// TIA Portal V20 export
TYPE "typeSafetyForcedDoorOpen"
// stored: Access Published, IsFailsafeCompliant true, Namespace Safety
   STRUCT
      Door1OpenMemo : Bool;
      Door2OpenMemo : Bool;
      Door3OpenMemo : Bool;
      Door4OpenMemo : Bool;
      Door5OpenMemo : Bool;
      Door6OpenMemo : Bool;
      Door7OpenMemo : Bool;
      Door8OpenMemo : Bool;
      Door9OpenMemo : Bool;
      Door10OpenMemo : Bool;
      Door1OpenMemoError : Bool;   // Forced Open AUTO SPLICE DOOR
      Door2OpenMemoError : Bool;   // Forced Open UNWIND MAIN DOOR
      Door3OpenMemoError : Bool;   // Forced Open UNWID TOP DOOR
      Door4OpenMemoError : Bool;   // Forced Open UNWIND BOTTOM DOOR
      Door5OpenMemoError : Bool;   // Forced Open STACK TABLE DOOR
      Door6OpenMemoError : Bool;   // Forced Open JR WINDER DOOR
      Door7OpenMemoError : Bool;   // Forced Open ANODE WASTE DOOR
      Door8OpenMemoError : Bool;   // Forced Open STACK TABLE REAR
      Door9OpenMemoError : Bool;   // Forced Open CATHODE WASTE DOOR
      Door10OpenMemoError : Bool;   // Forced Open UNWIND REAR DOOR
      Door1OpenTimeOver : Bool;   // Time Over Open AUTO SPLICE DOOR
      Door2OpenTimeOver : Bool;   // Time Over Open UNWIND MAIN DOOR
      Door3OpenTimeOver : Bool;   // Time Over Open UNWID TOP DOOR
      Door4OpenTimeOver : Bool;   // Time Over Open UNWIND BOTTOM DOOR
      Door5OpenTimeOver : Bool;   // Time Over Open STACK TABLE DOOR
      Door6OpenTimeOver : Bool;   // Time Over Open JR WINDER DOOR
      Door7OpenTimeOver : Bool;   // Time Over Open ANODE WASTE DOOR
      Door8OpenTimeOver : Bool;   // Time Over Open STACK TABLE REAR
      Door9OpenTimeOver : Bool;   // Time Over Open CATHODE WASTE DOOR
      Door10OpenTimeOver : Bool;   // Time Over Close UNWIND REAR DOOR
      Door1CloseTimeOver : Bool;   // Time Over Close AUTO SPLICE DOOR
      Door2CloseTimeOver : Bool;   // Time Over Close UNWIND MAIN DOOR
      Door3CloseTimeOver : Bool;   // Time Over Close UNWID TOP DOOR
      Door4CloseTimeOver : Bool;   // Time Over Close UNWIND BOTTOM DOOR
      Door5CloseTimeOver : Bool;   // Time Over Close STACK TABLE DOOR
      Door6CloseTimeOver : Bool;   // Time Over Close JR WINDER DOOR
      Door7CloseTimeOver : Bool;   // Time Over Close ANODE WASTE DOOR
      Door8CloseTimeOver : Bool;   // Time Over Close STACK TABLE REAR
      Door9CloseTimeOver : Bool;   // Time Over Close CATHODE WASTE DOOR
      Door10CloseTimeOver : Bool;   // Time Over Close UNWIND REAR DOOR
   END_STRUCT;
END_TYPE
